// Verify that all Switchbox valves are closed
FUNCTION F_SBVentInterlock : BOOL
VAR_INPUT
END_VAR
VAR
	stExpValveStatus : ST_SBValveStatuses := (
		bGateValveOpen:= FALSE, 
		bVentValveOpen:= FALSE, 
		bORingPumpValveOpen:= FALSE, 
		bForelineValveOpen:= FALSE, 
		bSlowPumpValveOpen:= FALSE,
		bSBVentOpen:= NOT GVL_BTS_VAC.fb_VP_VVC_1.q_xOPN_DO,
		bSBSlowVentOpen:= NOT GVL_BTS_VAC.fb_VP_VVC_2.q_xOPN_DO);
END_VAR

F_SBVentInterlock := F_VerifySBValveStatuses(stExpStatus := stExpValveStatus, bEnforce := FALSE);

END_FUNCTION

(* stored: Version 1.1.0.1, ProductVersion 3.1.4022.18
   POU F_SBVentInterlock: Id {2fc3d28b-9e53-4413-b140-bcabfe291b99}, SpecialFunc None *)
